FUNCTION_BLOCK DATA_SIMULATOR
  {SET_ATTRIBUTE(OpcUa, DEVICE.SENSOR)}
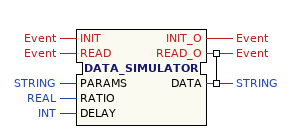
  EVENT_INPUT
    INIT;
    READ;
  END_EVENT
  EVENT_OUTPUT
    INIT_O;
    READ_O WITH DATA;
  END_EVENT
  VAR_INPUT
    PARAMS : STRING;
    RATIO : REAL;
    DELAY : INT;
  END_VAR
  VAR_OUTPUT
    DATA : STRING;
  END_VAR
END_FUNCTION_BLOCK
